TYPE ST_HMI_InOut :
STRUCT
	/// HMI direct (IN/OUT) struct
	/// e.g. for accessing (r/w) project specific settings

	//stM001 	: ST_M001_HMI_InOut;
	
	stSt010		: ST_St010_HMI_IN_OUT;
	stSt020		: ST_St020_HMI_IN_OUT;
	stSt030		: ST_St030_HMI_IN_OUT;
	stSt040		: ST_St040_HMI_IN_OUT;
	
	// global axis manager
	stHmiAxisManager	: ST_HmiAxisManager;
END_STRUCT
END_TYPE

(* stored: Version 1.1.0.1
   DUT ST_HMI_InOut: Id {169be2de-900d-4f38-8c5b-95d61db32dc2} *)
